{attribute 'linkalways'} 
{attribute 'no_explicit_call' := 'This FB is a CLASS and must be accessed using methods or properties'}
{attribute 'enable_dynamic_creation'}
FUNCTION_BLOCK FINAL MUL_LINT EXTENDS Node
VAR
	in1 : _LINT(0);
	in2 : _LINT(0);
	out : _LINT(0);
END_VAR

METHOD PUBLIC Clone : I_Node
VAR
	pNode : POINTER TO MUL_LINT;
END_VAR
pNode := __NEW(MUL_LINT);
Clone := pNode^;
END_METHOD

METHOD FB_init : BOOL
VAR_INPUT
	bInitRetains : BOOL; // if TRUE, the retain variables are initialized (warm start / cold start)
	bInCopyCode : BOOL;  // if TRUE, the instance afterwards gets moved into the copy code (online change)
END_VAR
AddInput('in1',THIS^.in1);
AddInput('in2',THIS^.in2);
AddOutput('out', THIS^.out);
END_METHOD

METHOD PROTECTED OnExecute
VAR
END_VAR
out.Value := in1.Value * in2.Value;
END_METHOD

END_FUNCTION_BLOCK

(* stored: Version 1.1.0.1, ProductVersion 3.1.4024.15
   POU MUL_LINT: Id {75f7e57c-c203-4e79-aac0-5ea38d5b469f}, SpecialFunc None
   Folder Constructor: Id {90d7faed-4cd2-437b-9bb0-3175d1577737}
   Method Clone: Id {73906c99-6afe-4778-b3ce-0615be73f6ea}
   Method FB_init: Id {d5b3b5e2-c0ab-49ef-a769-09c38613b3ee}
   Method OnExecute: Id {f9e66dd8-e8e6-4f67-b636-137dfba015ac} *)
